(* PLC project PLCOpen_Leer.project, CODESYS CODESYS V3.5 SP7 Patch 2 *)
(* stored: creationDateTime 2018-07-08T13:58:46.9898301, modificationDateTime 2018-07-08T13:57:47.963454 *)

VAR_GLOBAL  (* Global_GrafcetVars *)
  actStep_1 : BOOL := false;
  deactStep_1 : BOOL := false;
  Step_1 : BOOL := false;
  actStep_2 : BOOL := false;
  deactStep_2 : BOOL := false;
  Step_2 : BOOL := false;
  actEncStep_3 : BOOL := false;
  deactEncStep_3 : BOOL := false;
  EncStep_3 : BOOL := false;
  actEncStep_4 : BOOL := false;
  deactEncStep_4 : BOOL := false;
  EncStep_4 : BOOL := false;
  actStep_10 : BOOL := false;
  deactStep_10 : BOOL := false;
  Step_10 : BOOL := false;
  actEncStep_11 : BOOL := false;
  deactEncStep_11 : BOOL := false;
  EncStep_11 : BOOL := false;
  actEncStep_12 : BOOL := false;
  deactEncStep_12 : BOOL := false;
  EncStep_12 : BOOL := false;
  actEncStep_13 : BOOL := false;
  deactEncStep_13 : BOOL := false;
  EncStep_13 : BOOL := false;
  actEncStep_14 : BOOL := false;
  deactEncStep_14 : BOOL := false;
  EncStep_14 : BOOL := false;
  actEncStep_15 : BOOL := false;
  deactEncStep_15 : BOOL := false;
  EncStep_15 : BOOL := false;
  actEncStep_16 : BOOL := false;
  deactEncStep_16 : BOOL := false;
  EncStep_16 : BOOL := false;
  actStep_17 : BOOL := false;
  deactStep_17 : BOOL := false;
  Step_17 : BOOL := false;
  actStep_18 : BOOL := false;
  deactStep_18 : BOOL := false;
  Step_18 : BOOL := false;
  actStep_19 : BOOL := false;
  deactStep_19 : BOOL := false;
  Step_19 : BOOL := false;
  actStep_20 : BOOL := false;
  deactStep_20 : BOOL := false;
  Step_20 : BOOL := false;
  actStep_21 : BOOL := false;
  deactStep_21 : BOOL := false;
  Step_21 : BOOL := false;
  actStep_22 : BOOL := false;
  deactStep_22 : BOOL := false;
  Step_22 : BOOL := false;
  actStep_101 : BOOL := false;
  deactStep_101 : BOOL := false;
  Step_101 : BOOL := false;
  actStep_102 : BOOL := false;
  deactStep_102 : BOOL := false;
  Step_102 : BOOL := false;
  actStep_103 : BOOL := false;
  deactStep_103 : BOOL := false;
  Step_103 : BOOL := false;
  actStep_104 : BOOL := false;
  deactStep_104 : BOOL := false;
  Step_104 : BOOL := false;
  actStep_105 : BOOL := false;
  deactStep_105 : BOOL := false;
  Step_105 : BOOL := false;
  actStep_106 : BOOL := false;
  deactStep_106 : BOOL := false;
  Step_106 : BOOL := false;
  actStep_107 : BOOL := false;
  deactStep_107 : BOOL := false;
  Step_107 : BOOL := false;
  actStep_108 : BOOL := false;
  deactStep_108 : BOOL := false;
  Step_108 : BOOL := false;
  actStep_109 : BOOL := false;
  deactStep_109 : BOOL := false;
  Step_109 : BOOL := false;
  actStep_110 : BOOL := false;
  deactStep_110 : BOOL := false;
  Step_110 : BOOL := false;
  actStep_201 : BOOL := false;
  deactStep_201 : BOOL := false;
  Step_201 : BOOL := false;
  actStep_202 : BOOL := false;
  deactStep_202 : BOOL := false;
  Step_202 : BOOL := false;
  actStep_203 : BOOL := false;
  deactStep_203 : BOOL := false;
  Step_203 : BOOL := false;
  actStep_204 : BOOL := false;
  deactStep_204 : BOOL := false;
  Step_204 : BOOL := false;
  actStep_301 : BOOL := false;
  deactStep_301 : BOOL := false;
  Step_301 : BOOL := false;
  actStep_302 : BOOL := false;
  deactStep_302 : BOOL := false;
  Step_302 : BOOL := false;
  actStep_303 : BOOL := false;
  deactStep_303 : BOOL := false;
  Step_303 : BOOL := false;
  actStep_304 : BOOL := false;
  deactStep_304 : BOOL := false;
  Step_304 : BOOL := false;
  actStep_305 : BOOL := false;
  deactStep_305 : BOOL := false;
  Step_305 : BOOL := false;
  actStep_306 : BOOL := false;
  deactStep_306 : BOOL := false;
  Step_306 : BOOL := false;
  actStep_501 : BOOL := false;
  deactStep_501 : BOOL := false;
  Step_501 : BOOL := false;
  actStep_502 : BOOL := false;
  deactStep_502 : BOOL := false;
  Step_502 : BOOL := false;
  actStep_503 : BOOL := false;
  deactStep_503 : BOOL := false;
  Step_503 : BOOL := false;
  actStep_504 : BOOL := false;
  deactStep_504 : BOOL := false;
  Step_504 : BOOL := false;
  actStep_505 : BOOL := false;
  deactStep_505 : BOOL := false;
  Step_505 : BOOL := false;
  actStep_506 : BOOL := false;
  deactStep_506 : BOOL := false;
  Step_506 : BOOL := false;
  actStep_507 : BOOL := false;
  deactStep_507 : BOOL := false;
  Step_507 : BOOL := false;
  actStep_508 : BOOL := false;
  deactStep_508 : BOOL := false;
  Step_508 : BOOL := false;
  actStep_509 : BOOL := false;
  deactStep_509 : BOOL := false;
  Step_509 : BOOL := false;
  actStep_510 : BOOL := false;
  deactStep_510 : BOOL := false;
  Step_510 : BOOL := false;
  actStep_511 : BOOL := false;
  deactStep_511 : BOOL := false;
  Step_511 : BOOL := false;
  actStep_512 : BOOL := false;
  deactStep_512 : BOOL := false;
  Step_512 : BOOL := false;
  actStep_513 : BOOL := false;
  deactStep_513 : BOOL := false;
  Step_513 : BOOL := false;
  actStep_601 : BOOL := false;
  deactStep_601 : BOOL := false;
  Step_601 : BOOL := false;
  actStep_602 : BOOL := false;
  deactStep_602 : BOOL := false;
  Step_602 : BOOL := false;
  actStep_603 : BOOL := false;
  deactStep_603 : BOOL := false;
  Step_603 : BOOL := false;
  actStep_701 : BOOL := false;
  deactStep_701 : BOOL := false;
  Step_701 : BOOL := false;
  actStep_702 : BOOL := false;
  deactStep_702 : BOOL := false;
  Step_702 : BOOL := false;
  actStep_703 : BOOL := false;
  deactStep_703 : BOOL := false;
  Step_703 : BOOL := false;
  actStep_704 : BOOL := false;
  deactStep_704 : BOOL := false;
  Step_704 : BOOL := false;
  actStep_705 : BOOL := false;
  deactStep_705 : BOOL := false;
  Step_705 : BOOL := false;
  actStep_706 : BOOL := false;
  deactStep_706 : BOOL := false;
  Step_706 : BOOL := false;
  actStep_707 : BOOL := false;
  deactStep_707 : BOOL := false;
  Step_707 : BOOL := false;
  actStep_708 : BOOL := false;
  deactStep_708 : BOOL := false;
  Step_708 : BOOL := false;
  actStep_709 : BOOL := false;
  deactStep_709 : BOOL := false;
  Step_709 : BOOL := false;
  actStep_710 : BOOL := false;
  deactStep_710 : BOOL := false;
  Step_710 : BOOL := false;
  actStep_711 : BOOL := false;
  deactStep_711 : BOOL := false;
  Step_711 : BOOL := false;
  Foerderband : BOOL := false;
  Motorschutzschalter : BOOL := false;
  NOTAUS : BOOL := false;
  TellerAutomatik : BOOL := false;
  TellerHand : BOOL := false;
  Start : BOOL := false;
  Stopp : BOOL := false;
  TellerInPosition : BOOL := false;
  TellerDreht : BOOL := false;
  StartTeller : BOOL := false;
  Station1_fertig : BOOL := false;
  Station2_fertig : BOOL := false;
  Station3_fertig : BOOL := false;
  Station5_fertig : BOOL := false;
  Station6_fertig : BOOL := false;
  Station7_fertig : BOOL := false;
  TeilInVereinzelung1 : BOOL := false;
  TeilEingelaufen1 : BOOL := false;
  LinearVorne1 : BOOL := false;
  HandlingUnten1 : BOOL := false;
  ZangeZu1 : BOOL := false;
  HandlingOben1 : BOOL := false;
  LinearHinten1 : BOOL := false;
  ZangeAuf1 : BOOL := false;
  Lineareinheit1 : BOOL := false;
  Vereinzelung1 : BOOL := false;
  VorVereinzelung1 : BOOL := false;
  Handling1 : BOOL := false;
  Zange1 : BOOL := false;
  EindrueckenOben2 : BOOL := false;
  EindrueckenUnten2 : BOOL := false;
  StoerungQuittiert : BOOL := false;
  Stoerung2 : BOOL := false;
  K2 : INT := 0;
  Eindruecken2 : BOOL := false;
  2s/X202 : BOOL := false;
  SpannenOben3 : BOOL := false;
  SpannenUnten3 : BOOL := false;
  AusloeserVorne3 : BOOL := false;
  AusloeserHinten3 : BOOL := false;
  StoesselOben3 : BOOL := false;
  StoesselUnten3 : BOOL := false;
  Spannen3 : BOOL := false;
  Ausloeser3 : BOOL := false;
  Stoessel3 : BOOL := false;
  K3 : INT := 0;
  AusloeserHinten5 : BOOL := false;
  AusloeserVorne5 : BOOL := false;
  SpannenOben5 : BOOL := false;
  SpannenUnten5 : BOOL := false;
  StoesselOben5 : BOOL := false;
  StoesselUnten5 : BOOL := false;
  Kontrolle1 : BOOL := false;
  Kontrolle2 : BOOL := false;
  Kontrolle_Fehler : BOOL := false;
  KontaktierungHinten5 : BOOL := false;
  KontaktierungVorne5 : BOOL := false;
  Spannen5 : BOOL := false;
  Stoessel5 : BOOL := false;
  Ausloeser5 : BOOL := false;
  Kontaktierung5 : BOOL := false;
  GUTTEIL : BOOL := false;
  K51 : INT := 0;
  K52 : INT := 0;
  StempelHinten6 : BOOL := false;
  StempelVorne6 : BOOL := false;
  StempelIn6 : BOOL := false;
  LinearVorne7 : BOOL := false;
  LinearHinten7 : BOOL := false;
  LinearInPos7 : BOOL := false;
  HandlingUnten7 : BOOL := false;
  HandlingOben7 : BOOL := false;
  ZangeZu7 : BOOL := false;
  ZangeAuf7 : BOOL := false;
  LineareinheitVor7 : BOOL := false;
  Handling7 : BOOL := false;
  Zange7 : BOOL := false;
  LineareinheitZur7 : BOOL := false;
  K71 : INT := 0;
  K72 : INT := 0;
END_VAR

VAR_GLOBAL  (* Global_GrafcetParts *)
  Global_Grafcet : Grafcet_Control;
  PartialGrafcet_GlobalGrafcet : GlobalGrafcet;
  PartialGrafcet_G0 : G0;
  PartialGrafcet_G1 : G1;
  PartialGrafcet_G2 : G2;
  PartialGrafcet_G3 : G3;
  PartialGrafcet_G5 : G5;
  PartialGrafcet_G6 : G6;
  PartialGrafcet_G7 : G7;
END_VAR

FUNCTION_BLOCK Grafcet_Control
  VAR_INPUT
    Enable : BOOL := false;
    Init : BOOL := false;
    End : BOOL := false;
  END_VAR
  VAR
    StableState : BOOL := false;
    TranLoops : INT := 0;
    NumTran : INT := 0;
  END_VAR

		  	  
		  		IF Init THEN
		  		END_IF
		  		IF End THEN
		  		END_IF
		  		IF (Enable) THEN
		  			TranLoops := (0);
		  			StableState := true;
		  			WHILE ((StableState)AND(TranLoops<NumTran)) DO
		  			StableState := false;
		  			TranLoops := (TranLoops+1);
		  			IF ((INIT=FALSE)AND(END=FALSE)) THEN
		  			END_IF
		  			END_WHILE;
		  		END_IF
		  		
		  	  
		  	
END_FUNCTION_BLOCK

FUNCTION_BLOCK GlobalGrafcet
  VAR_INPUT
    Enable : BOOL := false;
    Init : BOOL := false;
    End : BOOL := false;
    Activate : BOOL := false;
    Freeze : BOOL := false;
  END_VAR
  VAR
    StableState : BOOL := false;
    TranLoops : INT := 0;
    NumTran : INT := 8;
    T_1 : BOOL := false;
    T_2 : BOOL := false;
    T_3 : BOOL := false;
    T_5 : BOOL := false;
    T_6 : BOOL := false;
    T_4 : BOOL := false;
    T_8 : BOOL := false;
    T_7 : BOOL := false;
  END_VAR

		  	  
		  		IF Init THEN
		  			Step_1 := true;
		  			actStep_1 := false;
		  			deactStep_1 := false;
		  			Step_2 := false;
		  			actStep_2 := false;
		  			deactStep_2 := false;
		  			EncStep_3 := false;
		  			actEncStep_3 := false;
		  			deactEncStep_3 := false;
		  			EncStep_4 := false;
		  			actEncStep_4 := false;
		  			deactEncStep_4 := false;
		  		END_IF
		  		IF Activate THEN
		  			Step_1 := false;
		  			actStep_1 := false;
		  			deactStep_1 := false;
		  			Step_2 := false;
		  			actStep_2 := false;
		  			deactStep_2 := false;
		  			EncStep_3 := false;
		  			actEncStep_3 := false;
		  			deactEncStep_3 := false;
		  			EncStep_4 := false;
		  			actEncStep_4 := false;
		  			deactEncStep_4 := false;
		  		END_IF
		  		IF End THEN
		  			Step_1 := false;
		  			actStep_1 := false;
		  			deactStep_1 := false;
		  			Step_2 := false;
		  			actStep_2 := false;
		  			deactStep_2 := false;
		  			EncStep_3 := false;
		  			actEncStep_3 := false;
		  			deactEncStep_3 := false;
		  			EncStep_4 := false;
		  			actEncStep_4 := false;
		  			deactEncStep_4 := false;
		  		END_IF
		  		IF (Enable) THEN
		  			TranLoops := (0);
		  			StableState := true;
		  			WHILE ((StableState)AND(TranLoops<NumTran)) DO
		  			StableState := false;
		  			TranLoops := (TranLoops+1);
		  			IF ((INIT=FALSE)AND(END=FALSE)) THEN
		  				T_1 := (Step_1)AND(Freeze=FALSE);
		  				T_2 := (Step_2)AND(Freeze=FALSE);
		  				T_3 := (Step_2)AND(Freeze=FALSE);
		  				T_5 := (EncStep_3)AND(Freeze=FALSE);
		  				T_6 := (EncStep_3)AND(Freeze=FALSE);
		  				T_4 := (Step_2)AND(Freeze=FALSE);
		  				T_8 := (EncStep_4)AND(Freeze=FALSE);
		  				T_7 := (EncStep_4)AND(Freeze=FALSE);
		  				IF ((( NOT NOTAUS) AND ( NOT Motorschutzschalter))AND(T_1)) THEN
		  					StableState := true;
		  					Step_1 := false;
		  					actStep_1 := false;
		  					deactStep_1 := true;
		  					Step_2 := true;
		  					actStep_2 := true;
		  					deactStep_2 := false;
		  				END_IF
		  				IF ((Start AND (TellerAutomatik AND ( NOT TellerHand)))AND(T_2)) THEN
		  					StableState := true;
		  					Step_2 := false;
		  					actStep_2 := false;
		  					deactStep_2 := true;
		  					EncStep_3 := true;
		  					actEncStep_3 := true;
		  					deactEncStep_3 := false;
		  				END_IF
		  				IF ((Start AND (( NOT TellerAutomatik) AND TellerHand))AND(T_3)) THEN
		  					StableState := true;
		  					Step_2 := false;
		  					actStep_2 := false;
		  					deactStep_2 := true;
		  					EncStep_4 := true;
		  					actEncStep_4 := true;
		  					deactEncStep_4 := false;
		  				END_IF
		  				IF ((Stopp AND (TellerHand AND ( NOT NOTAUS)))AND(T_5)) THEN
		  					StableState := true;
		  					EncStep_3 := false;
		  					actEncStep_3 := false;
		  					deactEncStep_3 := true;
		  					Step_2 := true;
		  					actStep_2 := true;
		  					deactStep_2 := false;
		  				END_IF
		  				IF ((NOTAUS)AND(T_6)) THEN
		  					StableState := true;
		  					EncStep_3 := false;
		  					actEncStep_3 := false;
		  					deactEncStep_3 := true;
		  					Step_1 := true;
		  					actStep_1 := true;
		  					deactStep_1 := false;
		  				END_IF
		  				IF ((NOTAUS)AND(T_4)) THEN
		  					StableState := true;
		  					Step_2 := false;
		  					actStep_2 := false;
		  					deactStep_2 := true;
		  					Step_1 := true;
		  					actStep_1 := true;
		  					deactStep_1 := false;
		  				END_IF
		  				IF ((NOTAUS)AND(T_8)) THEN
		  					StableState := true;
		  					EncStep_4 := false;
		  					actEncStep_4 := false;
		  					deactEncStep_4 := true;
		  					Step_1 := true;
		  					actStep_1 := true;
		  					deactStep_1 := false;
		  				END_IF
		  				IF ((Stopp AND (TellerHand AND ( NOT NOTAUS)))AND(T_7)) THEN
		  					StableState := true;
		  					EncStep_4 := false;
		  					actEncStep_4 := false;
		  					deactEncStep_4 := true;
		  					Step_2 := true;
		  					actStep_2 := true;
		  					deactStep_2 := false;
		  				END_IF
		  			END_IF
		  			IF (actStep_1)OR(Step_1)OR(deactStep_1) THEN
		  				IF actStep_1 THEN
		  					actStep_1 := false;
		  					Foerderband := FALSE;
		  				END_IF
		  				IF Step_1 THEN
		  				END_IF
		  				IF deactStep_1 THEN
		  					deactStep_1 := false;
		  				END_IF
		  			END_IF
		  			IF (actStep_2)OR(Step_2)OR(deactStep_2) THEN
		  				IF actStep_2 THEN
		  					actStep_2 := false;
		  				END_IF
		  				IF Step_2 THEN
		  				END_IF
		  				IF deactStep_2 THEN
		  					deactStep_2 := false;
		  				END_IF
		  			END_IF
		  			IF (actEncStep_3)OR(EncStep_3)OR(deactEncStep_3) THEN
		  				IF actEncStep_3 THEN
		  					actEncStep_3 := false;
		  					PartialGrafcet_G0(Enable := false, Init := false, Activate := true, End := false);
		  				END_IF
		  				IF EncStep_3 THEN
		  					PartialGrafcet_G0(Enable := true, Init := false, Activate := false, End := false);
		  				END_IF
		  				IF deactEncStep_3 THEN
		  					deactEncStep_3 := false;
		  					PartialGrafcet_G0(Enable := false, Init := false, Activate := false, End := true);
		  				END_IF
		  			END_IF
		  			IF (actEncStep_4)OR(EncStep_4)OR(deactEncStep_4) THEN
		  				IF actEncStep_4 THEN
		  					actEncStep_4 := false;
		  				END_IF
		  				IF EncStep_4 THEN
		  				END_IF
		  				IF deactEncStep_4 THEN
		  					deactEncStep_4 := false;
		  				END_IF
		  			END_IF
		  			END_WHILE;
		  		END_IF
		  		
		  	  
		  	
END_FUNCTION_BLOCK

FUNCTION_BLOCK G0
  VAR_INPUT
    Enable : BOOL := false;
    Init : BOOL := false;
    End : BOOL := false;
    Activate : BOOL := false;
    Freeze : BOOL := false;
  END_VAR
  VAR
    StableState : BOOL := false;
    TranLoops : INT := 0;
    NumTran : INT := 8;
    T_10 : BOOL := false;
    T_11 : BOOL := false;
    T_12 : BOOL := false;
    T_13 : BOOL := false;
    T_14 : BOOL := false;
    T_15 : BOOL := false;
    T_16 : BOOL := false;
    T_17 : BOOL := false;
  END_VAR

		  	  
		  		IF Init THEN
		  			Step_10 := false;
		  			actStep_10 := false;
		  			deactStep_10 := false;
		  			EncStep_11 := false;
		  			actEncStep_11 := false;
		  			deactEncStep_11 := false;
		  			EncStep_12 := false;
		  			actEncStep_12 := false;
		  			deactEncStep_12 := false;
		  			EncStep_13 := false;
		  			actEncStep_13 := false;
		  			deactEncStep_13 := false;
		  			EncStep_14 := false;
		  			actEncStep_14 := false;
		  			deactEncStep_14 := false;
		  			EncStep_15 := false;
		  			actEncStep_15 := false;
		  			deactEncStep_15 := false;
		  			EncStep_16 := false;
		  			actEncStep_16 := false;
		  			deactEncStep_16 := false;
		  			Step_17 := false;
		  			actStep_17 := false;
		  			deactStep_17 := false;
		  			Step_18 := false;
		  			actStep_18 := false;
		  			deactStep_18 := false;
		  			Step_19 := false;
		  			actStep_19 := false;
		  			deactStep_19 := false;
		  			Step_20 := false;
		  			actStep_20 := false;
		  			deactStep_20 := false;
		  			Step_21 := false;
		  			actStep_21 := false;
		  			deactStep_21 := false;
		  			Step_22 := false;
		  			actStep_22 := false;
		  			deactStep_22 := false;
		  		END_IF
		  		IF Activate THEN
		  			Step_10 := true;
		  			actStep_10 := true;
		  			deactStep_10 := false;
		  			EncStep_11 := false;
		  			actEncStep_11 := false;
		  			deactEncStep_11 := false;
		  			EncStep_12 := false;
		  			actEncStep_12 := false;
		  			deactEncStep_12 := false;
		  			EncStep_13 := false;
		  			actEncStep_13 := false;
		  			deactEncStep_13 := false;
		  			EncStep_14 := false;
		  			actEncStep_14 := false;
		  			deactEncStep_14 := false;
		  			EncStep_15 := false;
		  			actEncStep_15 := false;
		  			deactEncStep_15 := false;
		  			EncStep_16 := false;
		  			actEncStep_16 := false;
		  			deactEncStep_16 := false;
		  			Step_17 := false;
		  			actStep_17 := false;
		  			deactStep_17 := false;
		  			Step_18 := false;
		  			actStep_18 := false;
		  			deactStep_18 := false;
		  			Step_19 := false;
		  			actStep_19 := false;
		  			deactStep_19 := false;
		  			Step_20 := false;
		  			actStep_20 := false;
		  			deactStep_20 := false;
		  			Step_21 := false;
		  			actStep_21 := false;
		  			deactStep_21 := false;
		  			Step_22 := false;
		  			actStep_22 := false;
		  			deactStep_22 := false;
		  		END_IF
		  		IF End THEN
		  			Step_10 := false;
		  			actStep_10 := false;
		  			deactStep_10 := false;
		  			EncStep_11 := false;
		  			actEncStep_11 := false;
		  			deactEncStep_11 := false;
		  			EncStep_12 := false;
		  			actEncStep_12 := false;
		  			deactEncStep_12 := false;
		  			EncStep_13 := false;
		  			actEncStep_13 := false;
		  			deactEncStep_13 := false;
		  			EncStep_14 := false;
		  			actEncStep_14 := false;
		  			deactEncStep_14 := false;
		  			EncStep_15 := false;
		  			actEncStep_15 := false;
		  			deactEncStep_15 := false;
		  			EncStep_16 := false;
		  			actEncStep_16 := false;
		  			deactEncStep_16 := false;
		  			Step_17 := false;
		  			actStep_17 := false;
		  			deactStep_17 := false;
		  			Step_18 := false;
		  			actStep_18 := false;
		  			deactStep_18 := false;
		  			Step_19 := false;
		  			actStep_19 := false;
		  			deactStep_19 := false;
		  			Step_20 := false;
		  			actStep_20 := false;
		  			deactStep_20 := false;
		  			Step_21 := false;
		  			actStep_21 := false;
		  			deactStep_21 := false;
		  			Step_22 := false;
		  			actStep_22 := false;
		  			deactStep_22 := false;
		  		END_IF
		  		IF (Enable) THEN
		  			TranLoops := (0);
		  			StableState := true;
		  			WHILE ((StableState)AND(TranLoops<NumTran)) DO
		  			StableState := false;
		  			TranLoops := (TranLoops+1);
		  			IF ((INIT=FALSE)AND(END=FALSE)) THEN
		  				T_10 := (Step_10)AND(Freeze=FALSE);
		  				T_11 := (EncStep_11)AND(Freeze=FALSE);
		  				T_12 := (EncStep_12)AND(Freeze=FALSE);
		  				T_13 := (EncStep_13)AND(Freeze=FALSE);
		  				T_14 := (EncStep_14)AND(Freeze=FALSE);
		  				T_15 := (EncStep_15)AND(Freeze=FALSE);
		  				T_16 := (EncStep_16)AND(Freeze=FALSE);
		  				T_17 := (Step_17)AND(Step_18)AND(Step_19)AND(Step_20)AND(Step_21)AND(Step_22)AND(Freeze=FALSE);
		  				IF ((TellerInPosition AND TellerDreht)AND(T_10)) THEN
		  					StableState := true;
		  					Step_10 := false;
		  					actStep_10 := false;
		  					deactStep_10 := true;
		  					EncStep_11 := true;
		  					actEncStep_11 := true;
		  					deactEncStep_11 := false;
		  					EncStep_12 := true;
		  					actEncStep_12 := true;
		  					deactEncStep_12 := false;
		  					EncStep_13 := true;
		  					actEncStep_13 := true;
		  					deactEncStep_13 := false;
		  					EncStep_14 := true;
		  					actEncStep_14 := true;
		  					deactEncStep_14 := false;
		  					EncStep_15 := true;
		  					actEncStep_15 := true;
		  					deactEncStep_15 := false;
		  					EncStep_16 := true;
		  					actEncStep_16 := true;
		  					deactEncStep_16 := false;
		  				END_IF
		  				IF ((Station1_fertig)AND(T_11)) THEN
		  					StableState := true;
		  					EncStep_11 := false;
		  					actEncStep_11 := false;
		  					deactEncStep_11 := true;
		  					Step_17 := true;
		  					actStep_17 := true;
		  					deactStep_17 := false;
		  				END_IF
		  				IF ((Station2_fertig)AND(T_12)) THEN
		  					StableState := true;
		  					EncStep_12 := false;
		  					actEncStep_12 := false;
		  					deactEncStep_12 := true;
		  					Step_18 := true;
		  					actStep_18 := true;
		  					deactStep_18 := false;
		  				END_IF
		  				IF ((Station3_fertig)AND(T_13)) THEN
		  					StableState := true;
		  					EncStep_13 := false;
		  					actEncStep_13 := false;
		  					deactEncStep_13 := true;
		  					Step_19 := true;
		  					actStep_19 := true;
		  					deactStep_19 := false;
		  				END_IF
		  				IF ((Station5_fertig)AND(T_14)) THEN
		  					StableState := true;
		  					EncStep_14 := false;
		  					actEncStep_14 := false;
		  					deactEncStep_14 := true;
		  					Step_20 := true;
		  					actStep_20 := true;
		  					deactStep_20 := false;
		  				END_IF
		  				IF ((Station6_fertig)AND(T_15)) THEN
		  					StableState := true;
		  					EncStep_15 := false;
		  					actEncStep_15 := false;
		  					deactEncStep_15 := true;
		  					Step_21 := true;
		  					actStep_21 := true;
		  					deactStep_21 := false;
		  				END_IF
		  				IF ((Station7_fertig)AND(T_16)) THEN
		  					StableState := true;
		  					EncStep_16 := false;
		  					actEncStep_16 := false;
		  					deactEncStep_16 := true;
		  					Step_22 := true;
		  					actStep_22 := true;
		  					deactStep_22 := false;
		  				END_IF
		  				IF (((Station1_fertig AND Station2_fertig) AND ((Station3_fertig AND Station5_fertig) AND (Station6_fertig AND Station7_fertig)))AND(T_17)) THEN
		  					StableState := true;
		  					Step_17 := false;
		  					actStep_17 := false;
		  					deactStep_17 := true;
		  					Step_18 := false;
		  					actStep_18 := false;
		  					deactStep_18 := true;
		  					Step_19 := false;
		  					actStep_19 := false;
		  					deactStep_19 := true;
		  					Step_20 := false;
		  					actStep_20 := false;
		  					deactStep_20 := true;
		  					Step_21 := false;
		  					actStep_21 := false;
		  					deactStep_21 := true;
		  					Step_22 := false;
		  					actStep_22 := false;
		  					deactStep_22 := true;
		  					Step_10 := true;
		  					actStep_10 := true;
		  					deactStep_10 := false;
		  				END_IF
		  			END_IF
		  			IF (actStep_10)OR(Step_10)OR(deactStep_10) THEN
		  				IF actStep_10 THEN
		  					actStep_10 := false;
		  					Foerderband := TRUE;
		  				END_IF
		  				IF Step_10 THEN
		  					StartTeller := true;
		  				END_IF
		  				IF deactStep_10 THEN
		  					deactStep_10 := false;
		  					StartTeller := false;
		  				END_IF
		  			END_IF
		  			IF (actEncStep_11)OR(EncStep_11)OR(deactEncStep_11) THEN
		  				IF actEncStep_11 THEN
		  					actEncStep_11 := false;
		  					PartialGrafcet_G1(Enable := false, Init := false, Activate := true, End := false);
		  				END_IF
		  				IF EncStep_11 THEN
		  					PartialGrafcet_G1(Enable := true, Init := false, Activate := false, End := false);
		  				END_IF
		  				IF deactEncStep_11 THEN
		  					deactEncStep_11 := false;
		  					PartialGrafcet_G1(Enable := false, Init := false, Activate := false, End := true);
		  				END_IF
		  			END_IF
		  			IF (actEncStep_12)OR(EncStep_12)OR(deactEncStep_12) THEN
		  				IF actEncStep_12 THEN
		  					actEncStep_12 := false;
		  					PartialGrafcet_G2(Enable := false, Init := false, Activate := true, End := false);
		  				END_IF
		  				IF EncStep_12 THEN
		  					PartialGrafcet_G2(Enable := true, Init := false, Activate := false, End := false);
		  				END_IF
		  				IF deactEncStep_12 THEN
		  					deactEncStep_12 := false;
		  					PartialGrafcet_G2(Enable := false, Init := false, Activate := false, End := true);
		  				END_IF
		  			END_IF
		  			IF (actEncStep_13)OR(EncStep_13)OR(deactEncStep_13) THEN
		  				IF actEncStep_13 THEN
		  					actEncStep_13 := false;
		  					PartialGrafcet_G3(Enable := false, Init := false, Activate := true, End := false);
		  				END_IF
		  				IF EncStep_13 THEN
		  					PartialGrafcet_G3(Enable := true, Init := false, Activate := false, End := false);
		  				END_IF
		  				IF deactEncStep_13 THEN
		  					deactEncStep_13 := false;
		  					PartialGrafcet_G3(Enable := false, Init := false, Activate := false, End := true);
		  				END_IF
		  			END_IF
		  			IF (actEncStep_14)OR(EncStep_14)OR(deactEncStep_14) THEN
		  				IF actEncStep_14 THEN
		  					actEncStep_14 := false;
		  					PartialGrafcet_G5(Enable := false, Init := false, Activate := true, End := false);
		  				END_IF
		  				IF EncStep_14 THEN
		  					PartialGrafcet_G5(Enable := true, Init := false, Activate := false, End := false);
		  				END_IF
		  				IF deactEncStep_14 THEN
		  					deactEncStep_14 := false;
		  					PartialGrafcet_G5(Enable := false, Init := false, Activate := false, End := true);
		  				END_IF
		  			END_IF
		  			IF (actEncStep_15)OR(EncStep_15)OR(deactEncStep_15) THEN
		  				IF actEncStep_15 THEN
		  					actEncStep_15 := false;
		  					PartialGrafcet_G5(Enable := false, Init := false, Activate := true, End := false);
		  				END_IF
		  				IF EncStep_15 THEN
		  					PartialGrafcet_G5(Enable := true, Init := false, Activate := false, End := false);
		  				END_IF
		  				IF deactEncStep_15 THEN
		  					deactEncStep_15 := false;
		  					PartialGrafcet_G5(Enable := false, Init := false, Activate := false, End := true);
		  				END_IF
		  			END_IF
		  			IF (actEncStep_16)OR(EncStep_16)OR(deactEncStep_16) THEN
		  				IF actEncStep_16 THEN
		  					actEncStep_16 := false;
		  					PartialGrafcet_G7(Enable := false, Init := false, Activate := true, End := false);
		  				END_IF
		  				IF EncStep_16 THEN
		  					PartialGrafcet_G7(Enable := true, Init := false, Activate := false, End := false);
		  				END_IF
		  				IF deactEncStep_16 THEN
		  					deactEncStep_16 := false;
		  					PartialGrafcet_G7(Enable := false, Init := false, Activate := false, End := true);
		  				END_IF
		  			END_IF
		  			IF (actStep_17)OR(Step_17)OR(deactStep_17) THEN
		  				IF actStep_17 THEN
		  					actStep_17 := false;
		  				END_IF
		  				IF Step_17 THEN
		  				END_IF
		  				IF deactStep_17 THEN
		  					deactStep_17 := false;
		  				END_IF
		  			END_IF
		  			IF (actStep_18)OR(Step_18)OR(deactStep_18) THEN
		  				IF actStep_18 THEN
		  					actStep_18 := false;
		  				END_IF
		  				IF Step_18 THEN
		  				END_IF
		  				IF deactStep_18 THEN
		  					deactStep_18 := false;
		  				END_IF
		  			END_IF
		  			IF (actStep_19)OR(Step_19)OR(deactStep_19) THEN
		  				IF actStep_19 THEN
		  					actStep_19 := false;
		  				END_IF
		  				IF Step_19 THEN
		  				END_IF
		  				IF deactStep_19 THEN
		  					deactStep_19 := false;
		  				END_IF
		  			END_IF
		  			IF (actStep_20)OR(Step_20)OR(deactStep_20) THEN
		  				IF actStep_20 THEN
		  					actStep_20 := false;
		  				END_IF
		  				IF Step_20 THEN
		  				END_IF
		  				IF deactStep_20 THEN
		  					deactStep_20 := false;
		  				END_IF
		  			END_IF
		  			IF (actStep_21)OR(Step_21)OR(deactStep_21) THEN
		  				IF actStep_21 THEN
		  					actStep_21 := false;
		  				END_IF
		  				IF Step_21 THEN
		  				END_IF
		  				IF deactStep_21 THEN
		  					deactStep_21 := false;
		  				END_IF
		  			END_IF
		  			IF (actStep_22)OR(Step_22)OR(deactStep_22) THEN
		  				IF actStep_22 THEN
		  					actStep_22 := false;
		  				END_IF
		  				IF Step_22 THEN
		  				END_IF
		  				IF deactStep_22 THEN
		  					deactStep_22 := false;
		  				END_IF
		  			END_IF
		  			END_WHILE;
		  		END_IF
		  		
		  	  
		  	
END_FUNCTION_BLOCK

FUNCTION_BLOCK G1
  VAR_INPUT
    Enable : BOOL := false;
    Init : BOOL := false;
    End : BOOL := false;
    Activate : BOOL := false;
    Freeze : BOOL := false;
  END_VAR
  VAR
    StableState : BOOL := false;
    TranLoops : INT := 0;
    NumTran : INT := 10;
    T_101 : BOOL := false;
    T_102 : BOOL := false;
    T_103 : BOOL := false;
    T_104 : BOOL := false;
    T_105 : BOOL := false;
    T_106 : BOOL := false;
    T_107 : BOOL := false;
    T_108 : BOOL := false;
    T_109 : BOOL := false;
    T_110 : BOOL := false;
  END_VAR

		  	  
		  		IF Init THEN
		  			Step_101 := false;
		  			actStep_101 := false;
		  			deactStep_101 := false;
		  			Step_102 := false;
		  			actStep_102 := false;
		  			deactStep_102 := false;
		  			Step_103 := false;
		  			actStep_103 := false;
		  			deactStep_103 := false;
		  			Step_104 := false;
		  			actStep_104 := false;
		  			deactStep_104 := false;
		  			Step_105 := false;
		  			actStep_105 := false;
		  			deactStep_105 := false;
		  			Step_106 := false;
		  			actStep_106 := false;
		  			deactStep_106 := false;
		  			Step_107 := false;
		  			actStep_107 := false;
		  			deactStep_107 := false;
		  			Step_108 := false;
		  			actStep_108 := false;
		  			deactStep_108 := false;
		  			Step_109 := false;
		  			actStep_109 := false;
		  			deactStep_109 := false;
		  			Step_110 := false;
		  			actStep_110 := false;
		  			deactStep_110 := false;
		  		END_IF
		  		IF Activate THEN
		  			Step_101 := false;
		  			actStep_101 := false;
		  			deactStep_101 := false;
		  			Step_102 := true;
		  			actStep_102 := true;
		  			deactStep_102 := false;
		  			Step_103 := false;
		  			actStep_103 := false;
		  			deactStep_103 := false;
		  			Step_104 := false;
		  			actStep_104 := false;
		  			deactStep_104 := false;
		  			Step_105 := false;
		  			actStep_105 := false;
		  			deactStep_105 := false;
		  			Step_106 := false;
		  			actStep_106 := false;
		  			deactStep_106 := false;
		  			Step_107 := false;
		  			actStep_107 := false;
		  			deactStep_107 := false;
		  			Step_108 := false;
		  			actStep_108 := false;
		  			deactStep_108 := false;
		  			Step_109 := false;
		  			actStep_109 := false;
		  			deactStep_109 := false;
		  			Step_110 := false;
		  			actStep_110 := false;
		  			deactStep_110 := false;
		  		END_IF
		  		IF End THEN
		  			Step_101 := false;
		  			actStep_101 := false;
		  			deactStep_101 := false;
		  			Step_102 := false;
		  			actStep_102 := false;
		  			deactStep_102 := false;
		  			Step_103 := false;
		  			actStep_103 := false;
		  			deactStep_103 := false;
		  			Step_104 := false;
		  			actStep_104 := false;
		  			deactStep_104 := false;
		  			Step_105 := false;
		  			actStep_105 := false;
		  			deactStep_105 := false;
		  			Step_106 := false;
		  			actStep_106 := false;
		  			deactStep_106 := false;
		  			Step_107 := false;
		  			actStep_107 := false;
		  			deactStep_107 := false;
		  			Step_108 := false;
		  			actStep_108 := false;
		  			deactStep_108 := false;
		  			Step_109 := false;
		  			actStep_109 := false;
		  			deactStep_109 := false;
		  			Step_110 := false;
		  			actStep_110 := false;
		  			deactStep_110 := false;
		  		END_IF
		  		IF (Enable) THEN
		  			TranLoops := (0);
		  			StableState := true;
		  			WHILE ((StableState)AND(TranLoops<NumTran)) DO
		  			StableState := false;
		  			TranLoops := (TranLoops+1);
		  			IF ((INIT=FALSE)AND(END=FALSE)) THEN
		  				T_101 := (Step_101)AND(Freeze=FALSE);
		  				T_102 := (Step_102)AND(Freeze=FALSE);
		  				T_103 := (Step_103)AND(Freeze=FALSE);
		  				T_104 := (Step_104)AND(Freeze=FALSE);
		  				T_105 := (Step_105)AND(Freeze=FALSE);
		  				T_106 := (Step_106)AND(Freeze=FALSE);
		  				T_107 := (Step_107)AND(Freeze=FALSE);
		  				T_108 := (Step_108)AND(Freeze=FALSE);
		  				T_109 := (Step_109)AND(Freeze=FALSE);
		  				T_110 := (Step_110)AND(Freeze=FALSE);
		  				IF ((TeilInVereinzelung1)AND(T_101)) THEN
		  					StableState := true;
		  					Step_101 := false;
		  					actStep_101 := false;
		  					deactStep_101 := true;
		  					Step_102 := true;
		  					actStep_102 := true;
		  					deactStep_102 := false;
		  				END_IF
		  				IF ((TeilEingelaufen1)AND(T_102)) THEN
		  					StableState := true;
		  					Step_102 := false;
		  					actStep_102 := false;
		  					deactStep_102 := true;
		  					Step_103 := true;
		  					actStep_103 := true;
		  					deactStep_103 := false;
		  				END_IF
		  				IF ((LinearVorne1)AND(T_103)) THEN
		  					StableState := true;
		  					Step_103 := false;
		  					actStep_103 := false;
		  					deactStep_103 := true;
		  					Step_104 := true;
		  					actStep_104 := true;
		  					deactStep_104 := false;
		  				END_IF
		  				IF ((HandlingUnten1)AND(T_104)) THEN
		  					StableState := true;
		  					Step_104 := false;
		  					actStep_104 := false;
		  					deactStep_104 := true;
		  					Step_105 := true;
		  					actStep_105 := true;
		  					deactStep_105 := false;
		  				END_IF
		  				IF ((ZangeZu1)AND(T_105)) THEN
		  					StableState := true;
		  					Step_105 := false;
		  					actStep_105 := false;
		  					deactStep_105 := true;
		  					Step_106 := true;
		  					actStep_106 := true;
		  					deactStep_106 := false;
		  				END_IF
		  				IF ((HandlingOben1)AND(T_106)) THEN
		  					StableState := true;
		  					Step_106 := false;
		  					actStep_106 := false;
		  					deactStep_106 := true;
		  					Step_107 := true;
		  					actStep_107 := true;
		  					deactStep_107 := false;
		  				END_IF
		  				IF ((LinearHinten1)AND(T_107)) THEN
		  					StableState := true;
		  					Step_107 := false;
		  					actStep_107 := false;
		  					deactStep_107 := true;
		  					Step_108 := true;
		  					actStep_108 := true;
		  					deactStep_108 := false;
		  				END_IF
		  				IF ((HandlingUnten1)AND(T_108)) THEN
		  					StableState := true;
		  					Step_108 := false;
		  					actStep_108 := false;
		  					deactStep_108 := true;
		  					Step_109 := true;
		  					actStep_109 := true;
		  					deactStep_109 := false;
		  				END_IF
		  				IF ((ZangeAuf1)AND(T_109)) THEN
		  					StableState := true;
		  					Step_109 := false;
		  					actStep_109 := false;
		  					deactStep_109 := true;
		  					Step_110 := true;
		  					actStep_110 := true;
		  					deactStep_110 := false;
		  				END_IF
		  				IF ((HandlingOben1)AND(T_110)) THEN
		  					StableState := true;
		  					Step_110 := false;
		  					actStep_110 := false;
		  					deactStep_110 := true;
		  					Step_101 := true;
		  					actStep_101 := true;
		  					deactStep_101 := false;
		  				END_IF
		  			END_IF
		  			IF (actStep_101)OR(Step_101)OR(deactStep_101) THEN
		  				IF actStep_101 THEN
		  					actStep_101 := false;
		  					Lineareinheit1 := TRUE;
		  					VorVereinzelung1 := TRUE;
		  					Vereinzelung1 := TRUE;
		  				END_IF
		  				IF Step_101 THEN
		  					Station1_fertig := true;
		  				END_IF
		  				IF deactStep_101 THEN
		  					deactStep_101 := false;
		  					Station1_fertig := false;
		  				END_IF
		  			END_IF
		  			IF (actStep_102)OR(Step_102)OR(deactStep_102) THEN
		  				IF actStep_102 THEN
		  					actStep_102 := false;
		  					Vereinzelung1 := FALSE;
		  					VorVereinzelung1 := FALSE;
		  				END_IF
		  				IF Step_102 THEN
		  				END_IF
		  				IF deactStep_102 THEN
		  					deactStep_102 := false;
		  				END_IF
		  			END_IF
		  			IF (actStep_103)OR(Step_103)OR(deactStep_103) THEN
		  				IF actStep_103 THEN
		  					actStep_103 := false;
		  					Vereinzelung1 := TRUE;
		  					VorVereinzelung1 := TRUE;
		  				END_IF
		  				IF Step_103 THEN
		  				END_IF
		  				IF deactStep_103 THEN
		  					deactStep_103 := false;
		  				END_IF
		  			END_IF
		  			IF (actStep_104)OR(Step_104)OR(deactStep_104) THEN
		  				IF actStep_104 THEN
		  					actStep_104 := false;
		  					Handling1 := TRUE;
		  				END_IF
		  				IF Step_104 THEN
		  				END_IF
		  				IF deactStep_104 THEN
		  					deactStep_104 := false;
		  				END_IF
		  			END_IF
		  			IF (actStep_105)OR(Step_105)OR(deactStep_105) THEN
		  				IF actStep_105 THEN
		  					actStep_105 := false;
		  					Zange1 := TRUE;
		  				END_IF
		  				IF Step_105 THEN
		  				END_IF
		  				IF deactStep_105 THEN
		  					deactStep_105 := false;
		  				END_IF
		  			END_IF
		  			IF (actStep_106)OR(Step_106)OR(deactStep_106) THEN
		  				IF actStep_106 THEN
		  					actStep_106 := false;
		  					Handling1 := FALSE;
		  				END_IF
		  				IF Step_106 THEN
		  				END_IF
		  				IF deactStep_106 THEN
		  					deactStep_106 := false;
		  				END_IF
		  			END_IF
		  			IF (actStep_107)OR(Step_107)OR(deactStep_107) THEN
		  				IF actStep_107 THEN
		  					actStep_107 := false;
		  					Lineareinheit1 := TRUE;
		  				END_IF
		  				IF Step_107 THEN
		  				END_IF
		  				IF deactStep_107 THEN
		  					deactStep_107 := false;
		  				END_IF
		  			END_IF
		  			IF (actStep_108)OR(Step_108)OR(deactStep_108) THEN
		  				IF actStep_108 THEN
		  					actStep_108 := false;
		  					Handling1 := TRUE;
		  				END_IF
		  				IF Step_108 THEN
		  				END_IF
		  				IF deactStep_108 THEN
		  					deactStep_108 := false;
		  				END_IF
		  			END_IF
		  			IF (actStep_109)OR(Step_109)OR(deactStep_109) THEN
		  				IF actStep_109 THEN
		  					actStep_109 := false;
		  					Zange1 := FALSE;
		  				END_IF
		  				IF Step_109 THEN
		  				END_IF
		  				IF deactStep_109 THEN
		  					deactStep_109 := false;
		  				END_IF
		  			END_IF
		  			IF (actStep_110)OR(Step_110)OR(deactStep_110) THEN
		  				IF actStep_110 THEN
		  					actStep_110 := false;
		  					Handling1 := FALSE;
		  				END_IF
		  				IF Step_110 THEN
		  				END_IF
		  				IF deactStep_110 THEN
		  					deactStep_110 := false;
		  				END_IF
		  			END_IF
		  			END_WHILE;
		  		END_IF
		  		
		  	  
		  	
END_FUNCTION_BLOCK

FUNCTION_BLOCK G2
  VAR_INPUT
    Enable : BOOL := false;
    Init : BOOL := false;
    End : BOOL := false;
    Activate : BOOL := false;
    Freeze : BOOL := false;
  END_VAR
  VAR
    StableState : BOOL := false;
    TranLoops : INT := 0;
    NumTran : INT := 6;
    T_201 : BOOL := false;
    T_202 : BOOL := false;
    T_206 : BOOL := false;
    T_203 : BOOL := false;
    T_204 : BOOL := false;
    T_205 : BOOL := false;
  END_VAR

		  	  
		  		IF Init THEN
		  			Step_201 := false;
		  			actStep_201 := false;
		  			deactStep_201 := false;
		  			Step_202 := false;
		  			actStep_202 := false;
		  			deactStep_202 := false;
		  			Step_203 := false;
		  			actStep_203 := false;
		  			deactStep_203 := false;
		  			Step_204 := false;
		  			actStep_204 := false;
		  			deactStep_204 := false;
		  		END_IF
		  		IF Activate THEN
		  			Step_201 := false;
		  			actStep_201 := false;
		  			deactStep_201 := false;
		  			Step_202 := true;
		  			actStep_202 := true;
		  			deactStep_202 := false;
		  			Step_203 := false;
		  			actStep_203 := false;
		  			deactStep_203 := false;
		  			Step_204 := false;
		  			actStep_204 := false;
		  			deactStep_204 := false;
		  		END_IF
		  		IF End THEN
		  			Step_201 := false;
		  			actStep_201 := false;
		  			deactStep_201 := false;
		  			Step_202 := false;
		  			actStep_202 := false;
		  			deactStep_202 := false;
		  			Step_203 := false;
		  			actStep_203 := false;
		  			deactStep_203 := false;
		  			Step_204 := false;
		  			actStep_204 := false;
		  			deactStep_204 := false;
		  		END_IF
		  		IF (Enable) THEN
		  			TranLoops := (0);
		  			StableState := true;
		  			WHILE ((StableState)AND(TranLoops<NumTran)) DO
		  			StableState := false;
		  			TranLoops := (TranLoops+1);
		  			IF ((INIT=FALSE)AND(END=FALSE)) THEN
		  				T_201 := (Step_201)AND(Freeze=FALSE);
		  				T_202 := (Step_202)AND(Freeze=FALSE);
		  				T_206 := (Step_202)AND(Freeze=FALSE);
		  				T_203 := (Step_203)AND(Freeze=FALSE);
		  				T_204 := (Step_203)AND(Freeze=FALSE);
		  				T_205 := (Step_204)AND(Freeze=FALSE);
		  				IF ((EindrueckenOben2)AND(T_201)) THEN
		  					StableState := true;
		  					Step_201 := false;
		  					actStep_201 := false;
		  					deactStep_201 := true;
		  					Step_202 := true;
		  					actStep_202 := true;
		  					deactStep_202 := false;
		  				END_IF
		  				IF ((( NOT EindrueckenOben2) AND 2s/X202)AND(T_202)) THEN
		  					StableState := true;
		  					Step_202 := false;
		  					actStep_202 := false;
		  					deactStep_202 := true;
		  					Step_203 := true;
		  					actStep_203 := true;
		  					deactStep_203 := false;
		  				END_IF
		  				IF ((EindrueckenUnten2 AND 2s/X202)AND(T_206)) THEN
		  					StableState := true;
		  					Step_202 := false;
		  					actStep_202 := false;
		  					deactStep_202 := true;
		  					Step_201 := true;
		  					actStep_201 := true;
		  					deactStep_201 := false;
		  				END_IF
		  				IF ((EindrueckenOben2 AND (K2 < 3))AND(T_203)) THEN
		  					StableState := true;
		  					Step_203 := false;
		  					actStep_203 := false;
		  					deactStep_203 := true;
		  					Step_201 := true;
		  					actStep_201 := true;
		  					deactStep_201 := false;
		  				END_IF
		  				IF ((EindrueckenOben2 AND (K2 = 3))AND(T_204)) THEN
		  					StableState := true;
		  					Step_203 := false;
		  					actStep_203 := false;
		  					deactStep_203 := true;
		  					Step_204 := true;
		  					actStep_204 := true;
		  					deactStep_204 := false;
		  				END_IF
		  				IF ((StoerungQuittiert)AND(T_205)) THEN
		  					StableState := true;
		  					Step_204 := false;
		  					actStep_204 := false;
		  					deactStep_204 := true;
		  					Step_201 := true;
		  					actStep_201 := true;
		  					deactStep_201 := false;
		  				END_IF
		  			END_IF
		  			IF (actStep_201)OR(Step_201)OR(deactStep_201) THEN
		  				IF actStep_201 THEN
		  					actStep_201 := false;
		  					K2 := 0;
		  				END_IF
		  				IF Step_201 THEN
		  					Station2_fertig := true;
		  				END_IF
		  				IF deactStep_201 THEN
		  					deactStep_201 := false;
		  					Station2_fertig := false;
		  				END_IF
		  			END_IF
		  			IF (actStep_202)OR(Step_202)OR(deactStep_202) THEN
		  				IF actStep_202 THEN
		  					actStep_202 := false;
		  				END_IF
		  				IF Step_202 THEN
		  					Eindruecken2 := true;
		  				END_IF
		  				IF deactStep_202 THEN
		  					deactStep_202 := false;
		  					Eindruecken2 := false;
		  				END_IF
		  			END_IF
		  			IF (actStep_203)OR(Step_203)OR(deactStep_203) THEN
		  				IF actStep_203 THEN
		  					actStep_203 := false;
		  					K2 := K2 + 1;
		  				END_IF
		  				IF Step_203 THEN
		  				END_IF
		  				IF deactStep_203 THEN
		  					deactStep_203 := false;
		  				END_IF
		  			END_IF
		  			IF (actStep_204)OR(Step_204)OR(deactStep_204) THEN
		  				IF actStep_204 THEN
		  					actStep_204 := false;
		  				END_IF
		  				IF Step_204 THEN
		  					Stoerung2 := true;
		  				END_IF
		  				IF deactStep_204 THEN
		  					deactStep_204 := false;
		  					Stoerung2 := false;
		  				END_IF
		  			END_IF
		  			END_WHILE;
		  		END_IF
		  		
		  	  
		  	
END_FUNCTION_BLOCK

FUNCTION_BLOCK G3
  VAR_INPUT
    Enable : BOOL := false;
    Init : BOOL := false;
    End : BOOL := false;
    Activate : BOOL := false;
    Freeze : BOOL := false;
  END_VAR
  VAR
    StableState : BOOL := false;
    TranLoops : INT := 0;
    NumTran : INT := 7;
    T_301 : BOOL := false;
    T_302 : BOOL := false;
    T_303 : BOOL := false;
    T_304 : BOOL := false;
    T_305 : BOOL := false;
    T_306 : BOOL := false;
    T_307 : BOOL := false;
  END_VAR

		  	  
		  		IF Init THEN
		  			Step_301 := false;
		  			actStep_301 := false;
		  			deactStep_301 := false;
		  			Step_302 := false;
		  			actStep_302 := false;
		  			deactStep_302 := false;
		  			Step_303 := false;
		  			actStep_303 := false;
		  			deactStep_303 := false;
		  			Step_304 := false;
		  			actStep_304 := false;
		  			deactStep_304 := false;
		  			Step_305 := false;
		  			actStep_305 := false;
		  			deactStep_305 := false;
		  			Step_306 := false;
		  			actStep_306 := false;
		  			deactStep_306 := false;
		  		END_IF
		  		IF Activate THEN
		  			Step_301 := false;
		  			actStep_301 := false;
		  			deactStep_301 := false;
		  			Step_302 := true;
		  			actStep_302 := true;
		  			deactStep_302 := false;
		  			Step_303 := false;
		  			actStep_303 := false;
		  			deactStep_303 := false;
		  			Step_304 := false;
		  			actStep_304 := false;
		  			deactStep_304 := false;
		  			Step_305 := false;
		  			actStep_305 := false;
		  			deactStep_305 := false;
		  			Step_306 := false;
		  			actStep_306 := false;
		  			deactStep_306 := false;
		  		END_IF
		  		IF End THEN
		  			Step_301 := false;
		  			actStep_301 := false;
		  			deactStep_301 := false;
		  			Step_302 := false;
		  			actStep_302 := false;
		  			deactStep_302 := false;
		  			Step_303 := false;
		  			actStep_303 := false;
		  			deactStep_303 := false;
		  			Step_304 := false;
		  			actStep_304 := false;
		  			deactStep_304 := false;
		  			Step_305 := false;
		  			actStep_305 := false;
		  			deactStep_305 := false;
		  			Step_306 := false;
		  			actStep_306 := false;
		  			deactStep_306 := false;
		  		END_IF
		  		IF (Enable) THEN
		  			TranLoops := (0);
		  			StableState := true;
		  			WHILE ((StableState)AND(TranLoops<NumTran)) DO
		  			StableState := false;
		  			TranLoops := (TranLoops+1);
		  			IF ((INIT=FALSE)AND(END=FALSE)) THEN
		  				T_301 := (Step_301)AND(Freeze=FALSE);
		  				T_302 := (Step_302)AND(Freeze=FALSE);
		  				T_303 := (Step_303)AND(Freeze=FALSE);
		  				T_304 := (Step_304)AND(Freeze=FALSE);
		  				T_305 := (Step_305)AND(Freeze=FALSE);
		  				T_306 := (Step_306)AND(Freeze=FALSE);
		  				T_307 := (Step_306)AND(Freeze=FALSE);
		  				IF ((SpannenOben3)AND(T_301)) THEN
		  					StableState := true;
		  					Step_301 := false;
		  					actStep_301 := false;
		  					deactStep_301 := true;
		  					Step_302 := true;
		  					actStep_302 := true;
		  					deactStep_302 := false;
		  				END_IF
		  				IF ((SpannenUnten3)AND(T_302)) THEN
		  					StableState := true;
		  					Step_302 := false;
		  					actStep_302 := false;
		  					deactStep_302 := true;
		  					Step_303 := true;
		  					actStep_303 := true;
		  					deactStep_303 := false;
		  				END_IF
		  				IF ((AusloeserVorne3)AND(T_303)) THEN
		  					StableState := true;
		  					Step_303 := false;
		  					actStep_303 := false;
		  					deactStep_303 := true;
		  					Step_304 := true;
		  					actStep_304 := true;
		  					deactStep_304 := false;
		  				END_IF
		  				IF ((StoesselUnten3)AND(T_304)) THEN
		  					StableState := true;
		  					Step_304 := false;
		  					actStep_304 := false;
		  					deactStep_304 := true;
		  					Step_305 := true;
		  					actStep_305 := true;
		  					deactStep_305 := false;
		  				END_IF
		  				IF ((StoesselOben3)AND(T_305)) THEN
		  					StableState := true;
		  					Step_305 := false;
		  					actStep_305 := false;
		  					deactStep_305 := true;
		  					Step_306 := true;
		  					actStep_306 := true;
		  					deactStep_306 := false;
		  				END_IF
		  				IF ((AusloeserHinten3 AND (K3 < 5))AND(T_306)) THEN
		  					StableState := true;
		  					Step_306 := false;
		  					actStep_306 := false;
		  					deactStep_306 := true;
		  					Step_303 := true;
		  					actStep_303 := true;
		  					deactStep_303 := false;
		  				END_IF
		  				IF ((AusloeserHinten3 AND (K3 = 0))AND(T_307)) THEN
		  					StableState := true;
		  					Step_306 := false;
		  					actStep_306 := false;
		  					deactStep_306 := true;
		  					Step_301 := true;
		  					actStep_301 := true;
		  					deactStep_301 := false;
		  				END_IF
		  			END_IF
		  			IF (actStep_301)OR(Step_301)OR(deactStep_301) THEN
		  				IF actStep_301 THEN
		  					actStep_301 := false;
		  					Spannen3 := FALSE;
		  					K3 := 0;
		  				END_IF
		  				IF Step_301 THEN
		  					Station3_fertig := true;
		  				END_IF
		  				IF deactStep_301 THEN
		  					deactStep_301 := false;
		  					Station3_fertig := false;
		  				END_IF
		  			END_IF
		  			IF (actStep_302)OR(Step_302)OR(deactStep_302) THEN
		  				IF actStep_302 THEN
		  					actStep_302 := false;
		  					Spannen3 := TRUE;
		  				END_IF
		  				IF Step_302 THEN
		  				END_IF
		  				IF deactStep_302 THEN
		  					deactStep_302 := false;
		  				END_IF
		  			END_IF
		  			IF (actStep_303)OR(Step_303)OR(deactStep_303) THEN
		  				IF actStep_303 THEN
		  					actStep_303 := false;
		  					Ausloeser3 := TRUE;
		  				END_IF
		  				IF Step_303 THEN
		  				END_IF
		  				IF deactStep_303 THEN
		  					deactStep_303 := false;
		  				END_IF
		  			END_IF
		  			IF (actStep_304)OR(Step_304)OR(deactStep_304) THEN
		  				IF actStep_304 THEN
		  					actStep_304 := false;
		  				END_IF
		  				IF Step_304 THEN
		  					Stoessel3 := true;
		  				END_IF
		  				IF deactStep_304 THEN
		  					deactStep_304 := false;
		  					Stoessel3 := false;
		  				END_IF
		  			END_IF
		  			IF (actStep_305)OR(Step_305)OR(deactStep_305) THEN
		  				IF actStep_305 THEN
		  					actStep_305 := false;
		  				END_IF
		  				IF Step_305 THEN
		  				END_IF
		  				IF deactStep_305 THEN
		  					deactStep_305 := false;
		  					Ausloeser3 := FALSE;
		  				END_IF
		  			END_IF
		  			IF (actStep_306)OR(Step_306)OR(deactStep_306) THEN
		  				IF actStep_306 THEN
		  					actStep_306 := false;
		  					K3 := K3 + 3;
		  				END_IF
		  				IF Step_306 THEN
		  				END_IF
		  				IF deactStep_306 THEN
		  					deactStep_306 := false;
		  				END_IF
		  			END_IF
		  			END_WHILE;
		  		END_IF
		  		
		  	  
		  	
END_FUNCTION_BLOCK

FUNCTION_BLOCK G5
  VAR_INPUT
    Enable : BOOL := false;
    Init : BOOL := false;
    End : BOOL := false;
    Activate : BOOL := false;
    Freeze : BOOL := false;
  END_VAR
  VAR
    StableState : BOOL := false;
    TranLoops : INT := 0;
    NumTran : INT := 15;
    T_501 : BOOL := false;
    T_502 : BOOL := false;
    T_503 : BOOL := false;
    T_504 : BOOL := false;
    T_505 : BOOL := false;
    T_506 : BOOL := false;
    T_507 : BOOL := false;
    T_508 : BOOL := false;
    T_509 : BOOL := false;
    T_510 : BOOL := false;
    T_511 : BOOL := false;
    T_512 : BOOL := false;
    T_513 : BOOL := false;
    T_514 : BOOL := false;
    T_515 : BOOL := false;
  END_VAR

		  	  
		  		IF Init THEN
		  			Step_501 := false;
		  			actStep_501 := false;
		  			deactStep_501 := false;
		  			Step_502 := false;
		  			actStep_502 := false;
		  			deactStep_502 := false;
		  			Step_503 := false;
		  			actStep_503 := false;
		  			deactStep_503 := false;
		  			Step_504 := false;
		  			actStep_504 := false;
		  			deactStep_504 := false;
		  			Step_505 := false;
		  			actStep_505 := false;
		  			deactStep_505 := false;
		  			Step_506 := false;
		  			actStep_506 := false;
		  			deactStep_506 := false;
		  			Step_507 := false;
		  			actStep_507 := false;
		  			deactStep_507 := false;
		  			Step_508 := false;
		  			actStep_508 := false;
		  			deactStep_508 := false;
		  			Step_509 := false;
		  			actStep_509 := false;
		  			deactStep_509 := false;
		  			Step_510 := false;
		  			actStep_510 := false;
		  			deactStep_510 := false;
		  			Step_511 := false;
		  			actStep_511 := false;
		  			deactStep_511 := false;
		  			Step_512 := false;
		  			actStep_512 := false;
		  			deactStep_512 := false;
		  			Step_513 := false;
		  			actStep_513 := false;
		  			deactStep_513 := false;
		  		END_IF
		  		IF Activate THEN
		  			Step_501 := false;
		  			actStep_501 := false;
		  			deactStep_501 := false;
		  			Step_502 := true;
		  			actStep_502 := true;
		  			deactStep_502 := false;
		  			Step_503 := false;
		  			actStep_503 := false;
		  			deactStep_503 := false;
		  			Step_504 := false;
		  			actStep_504 := false;
		  			deactStep_504 := false;
		  			Step_505 := false;
		  			actStep_505 := false;
		  			deactStep_505 := false;
		  			Step_506 := false;
		  			actStep_506 := false;
		  			deactStep_506 := false;
		  			Step_507 := false;
		  			actStep_507 := false;
		  			deactStep_507 := false;
		  			Step_508 := false;
		  			actStep_508 := false;
		  			deactStep_508 := false;
		  			Step_509 := false;
		  			actStep_509 := false;
		  			deactStep_509 := false;
		  			Step_510 := false;
		  			actStep_510 := false;
		  			deactStep_510 := false;
		  			Step_511 := false;
		  			actStep_511 := false;
		  			deactStep_511 := false;
		  			Step_512 := false;
		  			actStep_512 := false;
		  			deactStep_512 := false;
		  			Step_513 := false;
		  			actStep_513 := false;
		  			deactStep_513 := false;
		  		END_IF
		  		IF End THEN
		  			Step_501 := false;
		  			actStep_501 := false;
		  			deactStep_501 := false;
		  			Step_502 := false;
		  			actStep_502 := false;
		  			deactStep_502 := false;
		  			Step_503 := false;
		  			actStep_503 := false;
		  			deactStep_503 := false;
		  			Step_504 := false;
		  			actStep_504 := false;
		  			deactStep_504 := false;
		  			Step_505 := false;
		  			actStep_505 := false;
		  			deactStep_505 := false;
		  			Step_506 := false;
		  			actStep_506 := false;
		  			deactStep_506 := false;
		  			Step_507 := false;
		  			actStep_507 := false;
		  			deactStep_507 := false;
		  			Step_508 := false;
		  			actStep_508 := false;
		  			deactStep_508 := false;
		  			Step_509 := false;
		  			actStep_509 := false;
		  			deactStep_509 := false;
		  			Step_510 := false;
		  			actStep_510 := false;
		  			deactStep_510 := false;
		  			Step_511 := false;
		  			actStep_511 := false;
		  			deactStep_511 := false;
		  			Step_512 := false;
		  			actStep_512 := false;
		  			deactStep_512 := false;
		  			Step_513 := false;
		  			actStep_513 := false;
		  			deactStep_513 := false;
		  		END_IF
		  		IF (Enable) THEN
		  			TranLoops := (0);
		  			StableState := true;
		  			WHILE ((StableState)AND(TranLoops<NumTran)) DO
		  			StableState := false;
		  			TranLoops := (TranLoops+1);
		  			IF ((INIT=FALSE)AND(END=FALSE)) THEN
		  				T_501 := (Step_501)AND(Freeze=FALSE);
		  				T_502 := (Step_502)AND(Freeze=FALSE);
		  				T_503 := (Step_503)AND(Freeze=FALSE);
		  				T_504 := (Step_504)AND(Freeze=FALSE);
		  				T_505 := (Step_505)AND(Freeze=FALSE);
		  				T_506 := (Step_506)AND(Freeze=FALSE);
		  				T_507 := (Step_508)AND(Freeze=FALSE);
		  				T_508 := (Step_509)AND(Freeze=FALSE);
		  				T_509 := (Step_508)AND(Freeze=FALSE);
		  				T_510 := (Step_511)AND(Freeze=FALSE);
		  				T_511 := (Step_507)AND(Step_510)AND(Freeze=FALSE);
		  				T_512 := (Step_507)AND(Step_510)AND(Freeze=FALSE);
		  				T_513 := (Step_507)AND(Step_510)AND(Freeze=FALSE);
		  				T_514 := (Step_512)AND(Freeze=FALSE);
		  				T_515 := (Step_513)AND(Freeze=FALSE);
		  				IF ((SpannenOben5)AND(T_501)) THEN
		  					StableState := true;
		  					Step_501 := false;
		  					actStep_501 := false;
		  					deactStep_501 := true;
		  					Step_502 := true;
		  					actStep_502 := true;
		  					deactStep_502 := false;
		  				END_IF
		  				IF ((SpannenUnten5)AND(T_502)) THEN
		  					StableState := true;
		  					Step_502 := false;
		  					actStep_502 := false;
		  					deactStep_502 := true;
		  					Step_503 := true;
		  					actStep_503 := true;
		  					deactStep_503 := false;
		  					Step_508 := true;
		  					actStep_508 := true;
		  					deactStep_508 := false;
		  				END_IF
		  				IF ((AusloeserVorne5)AND(T_503)) THEN
		  					StableState := true;
		  					Step_503 := false;
		  					actStep_503 := false;
		  					deactStep_503 := true;
		  					Step_504 := true;
		  					actStep_504 := true;
		  					deactStep_504 := false;
		  				END_IF
		  				IF ((StoesselUnten5)AND(T_504)) THEN
		  					StableState := true;
		  					Step_504 := false;
		  					actStep_504 := false;
		  					deactStep_504 := true;
		  					Step_505 := true;
		  					actStep_505 := true;
		  					deactStep_505 := false;
		  				END_IF
		  				IF ((StoesselOben5)AND(T_505)) THEN
		  					StableState := true;
		  					Step_505 := false;
		  					actStep_505 := false;
		  					deactStep_505 := true;
		  					Step_506 := true;
		  					actStep_506 := true;
		  					deactStep_506 := false;
		  				END_IF
		  				IF ((AusloeserHinten5)AND(T_506)) THEN
		  					StableState := true;
		  					Step_506 := false;
		  					actStep_506 := false;
		  					deactStep_506 := true;
		  					Step_507 := true;
		  					actStep_507 := true;
		  					deactStep_507 := false;
		  				END_IF
		  				IF ((KontaktierungVorne5 AND (Kontrolle1 AND Kontrolle2))AND(T_507)) THEN
		  					StableState := true;
		  					Step_508 := false;
		  					actStep_508 := false;
		  					deactStep_508 := true;
		  					Step_509 := true;
		  					actStep_509 := true;
		  					deactStep_509 := false;
		  				END_IF
		  				IF ((KontaktierungHinten5)AND(T_508)) THEN
		  					StableState := true;
		  					Step_509 := false;
		  					actStep_509 := false;
		  					deactStep_509 := true;
		  					Step_510 := true;
		  					actStep_510 := true;
		  					deactStep_510 := false;
		  				END_IF
		  				IF ((Kontrolle_Fehler)AND(T_509)) THEN
		  					StableState := true;
		  					Step_508 := false;
		  					actStep_508 := false;
		  					deactStep_508 := true;
		  					Step_511 := true;
		  					actStep_511 := true;
		  					deactStep_511 := false;
		  				END_IF
		  				IF ((KontaktierungHinten5)AND(T_510)) THEN
		  					StableState := true;
		  					Step_511 := false;
		  					actStep_511 := false;
		  					deactStep_511 := true;
		  					Step_510 := true;
		  					actStep_510 := true;
		  					deactStep_510 := false;
		  				END_IF
		  				IF (((K51 < 5) AND (K52 < 5))AND(T_511)) THEN
		  					StableState := true;
		  					Step_507 := false;
		  					actStep_507 := false;
		  					deactStep_507 := true;
		  					Step_510 := false;
		  					actStep_510 := false;
		  					deactStep_510 := true;
		  					Step_502 := true;
		  					actStep_502 := true;
		  					deactStep_502 := false;
		  				END_IF
		  				IF (((K51 = 5) AND (K52 = 5))AND(T_512)) THEN
		  					StableState := true;
		  					Step_507 := false;
		  					actStep_507 := false;
		  					deactStep_507 := true;
		  					Step_510 := false;
		  					actStep_510 := false;
		  					deactStep_510 := true;
		  					Step_512 := true;
		  					actStep_512 := true;
		  					deactStep_512 := false;
		  				END_IF
		  				IF (((K51 = 5) AND (K52 < 5))AND(T_513)) THEN
		  					StableState := true;
		  					Step_507 := false;
		  					actStep_507 := false;
		  					deactStep_507 := true;
		  					Step_510 := false;
		  					actStep_510 := false;
		  					deactStep_510 := true;
		  					Step_513 := true;
		  					actStep_513 := true;
		  					deactStep_513 := false;
		  				END_IF
		  				IF ((TRUE)AND(T_514)) THEN
		  					StableState := true;
		  					Step_512 := false;
		  					actStep_512 := false;
		  					deactStep_512 := true;
		  					Step_501 := true;
		  					actStep_501 := true;
		  					deactStep_501 := false;
		  				END_IF
		  				IF ((TRUE)AND(T_515)) THEN
		  					StableState := true;
		  					Step_513 := false;
		  					actStep_513 := false;
		  					deactStep_513 := true;
		  					Step_501 := true;
		  					actStep_501 := true;
		  					deactStep_501 := false;
		  				END_IF
		  			END_IF
		  			IF (actStep_501)OR(Step_501)OR(deactStep_501) THEN
		  				IF actStep_501 THEN
		  					actStep_501 := false;
		  					K51 := 0;
		  					K52 := 0;
		  					Spannen5 := FALSE;
		  				END_IF
		  				IF Step_501 THEN
		  					Station5_fertig := true;
		  				END_IF
		  				IF deactStep_501 THEN
		  					deactStep_501 := false;
		  					Station5_fertig := false;
		  				END_IF
		  			END_IF
		  			IF (actStep_502)OR(Step_502)OR(deactStep_502) THEN
		  				IF actStep_502 THEN
		  					actStep_502 := false;
		  					Spannen5 := TRUE;
		  				END_IF
		  				IF Step_502 THEN
		  				END_IF
		  				IF deactStep_502 THEN
		  					deactStep_502 := false;
		  				END_IF
		  			END_IF
		  			IF (actStep_503)OR(Step_503)OR(deactStep_503) THEN
		  				IF actStep_503 THEN
		  					actStep_503 := false;
		  					Ausloeser5 := TRUE;
		  				END_IF
		  				IF Step_503 THEN
		  				END_IF
		  				IF deactStep_503 THEN
		  					deactStep_503 := false;
		  				END_IF
		  			END_IF
		  			IF (actStep_504)OR(Step_504)OR(deactStep_504) THEN
		  				IF actStep_504 THEN
		  					actStep_504 := false;
		  				END_IF
		  				IF Step_504 THEN
		  					Stoessel5 := true;
		  				END_IF
		  				IF deactStep_504 THEN
		  					deactStep_504 := false;
		  					Stoessel5 := false;
		  				END_IF
		  			END_IF
		  			IF (actStep_505)OR(Step_505)OR(deactStep_505) THEN
		  				IF actStep_505 THEN
		  					actStep_505 := false;
		  				END_IF
		  				IF Step_505 THEN
		  				END_IF
		  				IF deactStep_505 THEN
		  					deactStep_505 := false;
		  					Ausloeser5 := FALSE;
		  				END_IF
		  			END_IF
		  			IF (actStep_506)OR(Step_506)OR(deactStep_506) THEN
		  				IF actStep_506 THEN
		  					actStep_506 := false;
		  					K51 := K51 + 1;
		  				END_IF
		  				IF Step_506 THEN
		  				END_IF
		  				IF deactStep_506 THEN
		  					deactStep_506 := false;
		  				END_IF
		  			END_IF
		  			IF (actStep_507)OR(Step_507)OR(deactStep_507) THEN
		  				IF actStep_507 THEN
		  					actStep_507 := false;
		  				END_IF
		  				IF Step_507 THEN
		  				END_IF
		  				IF deactStep_507 THEN
		  					deactStep_507 := false;
		  				END_IF
		  			END_IF
		  			IF (actStep_508)OR(Step_508)OR(deactStep_508) THEN
		  				IF actStep_508 THEN
		  					actStep_508 := false;
		  					Kontaktierung5 := TRUE;
		  				END_IF
		  				IF Step_508 THEN
		  				END_IF
		  				IF deactStep_508 THEN
		  					deactStep_508 := false;
		  				END_IF
		  			END_IF
		  			IF (actStep_509)OR(Step_509)OR(deactStep_509) THEN
		  				IF actStep_509 THEN
		  					actStep_509 := false;
		  					Kontaktierung5 := FALSE;
		  					K52 := K52 + 1;
		  				END_IF
		  				IF Step_509 THEN
		  				END_IF
		  				IF deactStep_509 THEN
		  					deactStep_509 := false;
		  				END_IF
		  			END_IF
		  			IF (actStep_510)OR(Step_510)OR(deactStep_510) THEN
		  				IF actStep_510 THEN
		  					actStep_510 := false;
		  				END_IF
		  				IF Step_510 THEN
		  				END_IF
		  				IF deactStep_510 THEN
		  					deactStep_510 := false;
		  				END_IF
		  			END_IF
		  			IF (actStep_511)OR(Step_511)OR(deactStep_511) THEN
		  				IF actStep_511 THEN
		  					actStep_511 := false;
		  					Kontaktierung5 := FALSE;
		  				END_IF
		  				IF Step_511 THEN
		  				END_IF
		  				IF deactStep_511 THEN
		  					deactStep_511 := false;
		  				END_IF
		  			END_IF
		  			IF (actStep_512)OR(Step_512)OR(deactStep_512) THEN
		  				IF actStep_512 THEN
		  					actStep_512 := false;
		  					GUTTEIL := TRUE;
		  				END_IF
		  				IF Step_512 THEN
		  				END_IF
		  				IF deactStep_512 THEN
		  					deactStep_512 := false;
		  				END_IF
		  			END_IF
		  			IF (actStep_513)OR(Step_513)OR(deactStep_513) THEN
		  				IF actStep_513 THEN
		  					actStep_513 := false;
		  					GUTTEIL := FALSE;
		  				END_IF
		  				IF Step_513 THEN
		  				END_IF
		  				IF deactStep_513 THEN
		  					deactStep_513 := false;
		  				END_IF
		  			END_IF
		  			END_WHILE;
		  		END_IF
		  		
		  	  
		  	
END_FUNCTION_BLOCK

FUNCTION_BLOCK G6
  VAR_INPUT
    Enable : BOOL := false;
    Init : BOOL := false;
    End : BOOL := false;
    Activate : BOOL := false;
    Freeze : BOOL := false;
  END_VAR
  VAR
    StableState : BOOL := false;
    TranLoops : INT := 0;
    NumTran : INT := 3;
    T_601 : BOOL := false;
    T_602 : BOOL := false;
    T_603 : BOOL := false;
  END_VAR

		  	  
		  		IF Init THEN
		  			Step_601 := false;
		  			actStep_601 := false;
		  			deactStep_601 := false;
		  			Step_602 := false;
		  			actStep_602 := false;
		  			deactStep_602 := false;
		  			Step_603 := false;
		  			actStep_603 := false;
		  			deactStep_603 := false;
		  		END_IF
		  		IF Activate THEN
		  			Step_601 := false;
		  			actStep_601 := false;
		  			deactStep_601 := false;
		  			Step_602 := true;
		  			actStep_602 := true;
		  			deactStep_602 := false;
		  			Step_603 := false;
		  			actStep_603 := false;
		  			deactStep_603 := false;
		  		END_IF
		  		IF End THEN
		  			Step_601 := false;
		  			actStep_601 := false;
		  			deactStep_601 := false;
		  			Step_602 := false;
		  			actStep_602 := false;
		  			deactStep_602 := false;
		  			Step_603 := false;
		  			actStep_603 := false;
		  			deactStep_603 := false;
		  		END_IF
		  		IF (Enable) THEN
		  			TranLoops := (0);
		  			StableState := true;
		  			WHILE ((StableState)AND(TranLoops<NumTran)) DO
		  			StableState := false;
		  			TranLoops := (TranLoops+1);
		  			IF ((INIT=FALSE)AND(END=FALSE)) THEN
		  				T_601 := (Step_601)AND(Freeze=FALSE);
		  				T_602 := (Step_602)AND(Freeze=FALSE);
		  				T_603 := (Step_603)AND(Freeze=FALSE);
		  				IF ((StempelHinten6)AND(T_601)) THEN
		  					StableState := true;
		  					Step_601 := false;
		  					actStep_601 := false;
		  					deactStep_601 := true;
		  					Step_602 := true;
		  					actStep_602 := true;
		  					deactStep_602 := false;
		  				END_IF
		  				IF ((GUTTEIL)AND(T_602)) THEN
		  					StableState := true;
		  					Step_602 := false;
		  					actStep_602 := false;
		  					deactStep_602 := true;
		  					Step_603 := true;
		  					actStep_603 := true;
		  					deactStep_603 := false;
		  				END_IF
		  				IF ((StempelVorne6)AND(T_603)) THEN
		  					StableState := true;
		  					Step_603 := false;
		  					actStep_603 := false;
		  					deactStep_603 := true;
		  					Step_601 := true;
		  					actStep_601 := true;
		  					deactStep_601 := false;
		  				END_IF
		  			END_IF
		  			IF (actStep_601)OR(Step_601)OR(deactStep_601) THEN
		  				IF actStep_601 THEN
		  					actStep_601 := false;
		  				END_IF
		  				IF Step_601 THEN
		  					Station6_fertig := true;
		  				END_IF
		  				IF deactStep_601 THEN
		  					deactStep_601 := false;
		  					Station6_fertig := false;
		  				END_IF
		  			END_IF
		  			IF (actStep_602)OR(Step_602)OR(deactStep_602) THEN
		  				IF actStep_602 THEN
		  					actStep_602 := false;
		  				END_IF
		  				IF Step_602 THEN
		  				END_IF
		  				IF deactStep_602 THEN
		  					deactStep_602 := false;
		  				END_IF
		  			END_IF
		  			IF (actStep_603)OR(Step_603)OR(deactStep_603) THEN
		  				IF actStep_603 THEN
		  					actStep_603 := false;
		  				END_IF
		  				IF Step_603 THEN
		  					StempelIn6 := true;
		  				END_IF
		  				IF deactStep_603 THEN
		  					deactStep_603 := false;
		  					StempelIn6 := false;
		  				END_IF
		  			END_IF
		  			END_WHILE;
		  		END_IF
		  		
		  	  
		  	
END_FUNCTION_BLOCK

FUNCTION_BLOCK G7
  VAR_INPUT
    Enable : BOOL := false;
    Init : BOOL := false;
    End : BOOL := false;
    Activate : BOOL := false;
    Freeze : BOOL := false;
  END_VAR
  VAR
    StableState : BOOL := false;
    TranLoops : INT := 0;
    NumTran : INT := 12;
    T_701 : BOOL := false;
    T_702 : BOOL := false;
    T_703 : BOOL := false;
    T_704 : BOOL := false;
    T_705 : BOOL := false;
    T_706 : BOOL := false;
    T_707 : BOOL := false;
    T_708 : BOOL := false;
    T_709 : BOOL := false;
    T_710 : BOOL := false;
    T_711 : BOOL := false;
    T_712 : BOOL := false;
  END_VAR

		  	  
		  		IF Init THEN
		  			Step_701 := false;
		  			actStep_701 := false;
		  			deactStep_701 := false;
		  			Step_702 := false;
		  			actStep_702 := false;
		  			deactStep_702 := false;
		  			Step_703 := false;
		  			actStep_703 := false;
		  			deactStep_703 := false;
		  			Step_704 := false;
		  			actStep_704 := false;
		  			deactStep_704 := false;
		  			Step_705 := false;
		  			actStep_705 := false;
		  			deactStep_705 := false;
		  			Step_706 := false;
		  			actStep_706 := false;
		  			deactStep_706 := false;
		  			Step_707 := false;
		  			actStep_707 := false;
		  			deactStep_707 := false;
		  			Step_708 := false;
		  			actStep_708 := false;
		  			deactStep_708 := false;
		  			Step_709 := false;
		  			actStep_709 := false;
		  			deactStep_709 := false;
		  			Step_710 := false;
		  			actStep_710 := false;
		  			deactStep_710 := false;
		  			Step_711 := false;
		  			actStep_711 := false;
		  			deactStep_711 := false;
		  		END_IF
		  		IF Activate THEN
		  			Step_701 := false;
		  			actStep_701 := false;
		  			deactStep_701 := false;
		  			Step_702 := true;
		  			actStep_702 := true;
		  			deactStep_702 := false;
		  			Step_703 := false;
		  			actStep_703 := false;
		  			deactStep_703 := false;
		  			Step_704 := false;
		  			actStep_704 := false;
		  			deactStep_704 := false;
		  			Step_705 := false;
		  			actStep_705 := false;
		  			deactStep_705 := false;
		  			Step_706 := false;
		  			actStep_706 := false;
		  			deactStep_706 := false;
		  			Step_707 := false;
		  			actStep_707 := false;
		  			deactStep_707 := false;
		  			Step_708 := false;
		  			actStep_708 := false;
		  			deactStep_708 := false;
		  			Step_709 := false;
		  			actStep_709 := false;
		  			deactStep_709 := false;
		  			Step_710 := false;
		  			actStep_710 := false;
		  			deactStep_710 := false;
		  			Step_711 := false;
		  			actStep_711 := false;
		  			deactStep_711 := false;
		  		END_IF
		  		IF End THEN
		  			Step_701 := false;
		  			actStep_701 := false;
		  			deactStep_701 := false;
		  			Step_702 := false;
		  			actStep_702 := false;
		  			deactStep_702 := false;
		  			Step_703 := false;
		  			actStep_703 := false;
		  			deactStep_703 := false;
		  			Step_704 := false;
		  			actStep_704 := false;
		  			deactStep_704 := false;
		  			Step_705 := false;
		  			actStep_705 := false;
		  			deactStep_705 := false;
		  			Step_706 := false;
		  			actStep_706 := false;
		  			deactStep_706 := false;
		  			Step_707 := false;
		  			actStep_707 := false;
		  			deactStep_707 := false;
		  			Step_708 := false;
		  			actStep_708 := false;
		  			deactStep_708 := false;
		  			Step_709 := false;
		  			actStep_709 := false;
		  			deactStep_709 := false;
		  			Step_710 := false;
		  			actStep_710 := false;
		  			deactStep_710 := false;
		  			Step_711 := false;
		  			actStep_711 := false;
		  			deactStep_711 := false;
		  		END_IF
		  		IF (Enable) THEN
		  			TranLoops := (0);
		  			StableState := true;
		  			WHILE ((StableState)AND(TranLoops<NumTran)) DO
		  			StableState := false;
		  			TranLoops := (TranLoops+1);
		  			IF ((INIT=FALSE)AND(END=FALSE)) THEN
		  				T_701 := (Step_701)AND(Freeze=FALSE);
		  				T_702 := (Step_702)AND(Freeze=FALSE);
		  				T_703 := (Step_703)AND(Freeze=FALSE);
		  				T_704 := (Step_704)AND(Freeze=FALSE);
		  				T_705 := (Step_705)AND(Freeze=FALSE);
		  				T_706 := (Step_706)AND(Freeze=FALSE);
		  				T_707 := (Step_707)AND(Freeze=FALSE);
		  				T_708 := (Step_708)AND(Freeze=FALSE);
		  				T_709 := (Step_704)AND(Freeze=FALSE);
		  				T_710 := (Step_709)AND(Freeze=FALSE);
		  				T_711 := (Step_710)AND(Freeze=FALSE);
		  				T_712 := (Step_711)AND(Freeze=FALSE);
		  				IF ((LinearVorne7)AND(T_701)) THEN
		  					StableState := true;
		  					Step_701 := false;
		  					actStep_701 := false;
		  					deactStep_701 := true;
		  					Step_702 := true;
		  					actStep_702 := true;
		  					deactStep_702 := false;
		  				END_IF
		  				IF ((HandlingUnten7)AND(T_702)) THEN
		  					StableState := true;
		  					Step_702 := false;
		  					actStep_702 := false;
		  					deactStep_702 := true;
		  					Step_703 := true;
		  					actStep_703 := true;
		  					deactStep_703 := false;
		  				END_IF
		  				IF ((ZangeZu7)AND(T_703)) THEN
		  					StableState := true;
		  					Step_703 := false;
		  					actStep_703 := false;
		  					deactStep_703 := true;
		  					Step_704 := true;
		  					actStep_704 := true;
		  					deactStep_704 := false;
		  				END_IF
		  				IF ((HandlingOben7 AND GUTTEIL)AND(T_704)) THEN
		  					StableState := true;
		  					Step_704 := false;
		  					actStep_704 := false;
		  					deactStep_704 := true;
		  					Step_705 := true;
		  					actStep_705 := true;
		  					deactStep_705 := false;
		  				END_IF
		  				IF ((LinearHinten7)AND(T_705)) THEN
		  					StableState := true;
		  					Step_705 := false;
		  					actStep_705 := false;
		  					deactStep_705 := true;
		  					Step_706 := true;
		  					actStep_706 := true;
		  					deactStep_706 := false;
		  				END_IF
		  				IF ((HandlingUnten7)AND(T_706)) THEN
		  					StableState := true;
		  					Step_706 := false;
		  					actStep_706 := false;
		  					deactStep_706 := true;
		  					Step_707 := true;
		  					actStep_707 := true;
		  					deactStep_707 := false;
		  				END_IF
		  				IF ((ZangeAuf7)AND(T_707)) THEN
		  					StableState := true;
		  					Step_707 := false;
		  					actStep_707 := false;
		  					deactStep_707 := true;
		  					Step_708 := true;
		  					actStep_708 := true;
		  					deactStep_708 := false;
		  				END_IF
		  				IF ((HandlingOben7)AND(T_708)) THEN
		  					StableState := true;
		  					Step_708 := false;
		  					actStep_708 := false;
		  					deactStep_708 := true;
		  					Step_701 := true;
		  					actStep_701 := true;
		  					deactStep_701 := false;
		  				END_IF
		  				IF ((HandlingOben7 AND ( NOT GUTTEIL))AND(T_709)) THEN
		  					StableState := true;
		  					Step_704 := false;
		  					actStep_704 := false;
		  					deactStep_704 := true;
		  					Step_709 := true;
		  					actStep_709 := true;
		  					deactStep_709 := false;
		  				END_IF
		  				IF ((LinearInPos7)AND(T_710)) THEN
		  					StableState := true;
		  					Step_709 := false;
		  					actStep_709 := false;
		  					deactStep_709 := true;
		  					Step_710 := true;
		  					actStep_710 := true;
		  					deactStep_710 := false;
		  				END_IF
		  				IF ((ZangeAuf7)AND(T_711)) THEN
		  					StableState := true;
		  					Step_710 := false;
		  					actStep_710 := false;
		  					deactStep_710 := true;
		  					Step_711 := true;
		  					actStep_711 := true;
		  					deactStep_711 := false;
		  				END_IF
		  				IF ((LinearHinten7)AND(T_712)) THEN
		  					StableState := true;
		  					Step_711 := false;
		  					actStep_711 := false;
		  					deactStep_711 := true;
		  					Step_701 := true;
		  					actStep_701 := true;
		  					deactStep_701 := false;
		  				END_IF
		  			END_IF
		  			IF (actStep_701)OR(Step_701)OR(deactStep_701) THEN
		  				IF actStep_701 THEN
		  					actStep_701 := false;
		  				END_IF
		  				IF Step_701 THEN
		  					Station7_fertig := true;
		  					LineareinheitVor7 := true;
		  				END_IF
		  				IF deactStep_701 THEN
		  					deactStep_701 := false;
		  					Station7_fertig := false;
		  					LineareinheitVor7 := false;
		  				END_IF
		  			END_IF
		  			IF (actStep_702)OR(Step_702)OR(deactStep_702) THEN
		  				IF actStep_702 THEN
		  					actStep_702 := false;
		  					Handling7 := TRUE;
		  				END_IF
		  				IF Step_702 THEN
		  				END_IF
		  				IF deactStep_702 THEN
		  					deactStep_702 := false;
		  				END_IF
		  			END_IF
		  			IF (actStep_703)OR(Step_703)OR(deactStep_703) THEN
		  				IF actStep_703 THEN
		  					actStep_703 := false;
		  					Zange7 := TRUE;
		  				END_IF
		  				IF Step_703 THEN
		  				END_IF
		  				IF deactStep_703 THEN
		  					deactStep_703 := false;
		  				END_IF
		  			END_IF
		  			IF (actStep_704)OR(Step_704)OR(deactStep_704) THEN
		  				IF actStep_704 THEN
		  					actStep_704 := false;
		  					Handling7 := FALSE;
		  				END_IF
		  				IF Step_704 THEN
		  				END_IF
		  				IF deactStep_704 THEN
		  					deactStep_704 := false;
		  				END_IF
		  			END_IF
		  			IF (actStep_705)OR(Step_705)OR(deactStep_705) THEN
		  				IF actStep_705 THEN
		  					actStep_705 := false;
		  				END_IF
		  				IF Step_705 THEN
		  					LineareinheitZur7 := true;
		  				END_IF
		  				IF deactStep_705 THEN
		  					deactStep_705 := false;
		  					LineareinheitZur7 := false;
		  				END_IF
		  			END_IF
		  			IF (actStep_706)OR(Step_706)OR(deactStep_706) THEN
		  				IF actStep_706 THEN
		  					actStep_706 := false;
		  					Handling7 := TRUE;
		  				END_IF
		  				IF Step_706 THEN
		  				END_IF
		  				IF deactStep_706 THEN
		  					deactStep_706 := false;
		  				END_IF
		  			END_IF
		  			IF (actStep_707)OR(Step_707)OR(deactStep_707) THEN
		  				IF actStep_707 THEN
		  					actStep_707 := false;
		  					Zange7 := FALSE;
		  				END_IF
		  				IF Step_707 THEN
		  				END_IF
		  				IF deactStep_707 THEN
		  					deactStep_707 := false;
		  				END_IF
		  			END_IF
		  			IF (actStep_708)OR(Step_708)OR(deactStep_708) THEN
		  				IF actStep_708 THEN
		  					actStep_708 := false;
		  					Handling7 := FALSE;
		  					K71 := K71 + 1;
		  				END_IF
		  				IF Step_708 THEN
		  				END_IF
		  				IF deactStep_708 THEN
		  					deactStep_708 := false;
		  				END_IF
		  			END_IF
		  			IF (actStep_709)OR(Step_709)OR(deactStep_709) THEN
		  				IF actStep_709 THEN
		  					actStep_709 := false;
		  				END_IF
		  				IF Step_709 THEN
		  					LineareinheitZur7 := true;
		  				END_IF
		  				IF deactStep_709 THEN
		  					deactStep_709 := false;
		  					LineareinheitZur7 := false;
		  				END_IF
		  			END_IF
		  			IF (actStep_710)OR(Step_710)OR(deactStep_710) THEN
		  				IF actStep_710 THEN
		  					actStep_710 := false;
		  					Zange7 := FALSE;
		  				END_IF
		  				IF Step_710 THEN
		  				END_IF
		  				IF deactStep_710 THEN
		  					deactStep_710 := false;
		  				END_IF
		  			END_IF
		  			IF (actStep_711)OR(Step_711)OR(deactStep_711) THEN
		  				IF actStep_711 THEN
		  					actStep_711 := false;
		  					K72 := K72 + 0;
		  				END_IF
		  				IF Step_711 THEN
		  					LineareinheitZur7 := true;
		  				END_IF
		  				IF deactStep_711 THEN
		  					deactStep_711 := false;
		  					LineareinheitZur7 := false;
		  				END_IF
		  			END_IF
		  			END_WHILE;
		  		END_IF
		  		
		  	  
		  	
END_FUNCTION_BLOCK
